INTERFACE I_AsyncRpcCall EXTENDS I_Disposable

METHOD PUBLIC Call
VAR_INPUT
END_VAR
END_METHOD

END_INTERFACE

(* stored: Version 1.1.0.1, ProductVersion 3.1.4026.13
   Itf I_AsyncRpcCall: Id {07cb245e-e3d8-0775-00fa-d716c6b736a7}
   Method Call: Id {7bad1aba-f8a0-0fbc-312d-4796e3e6ee72} *)
